(*
    MCS2 Motion Stage
    Controls a stage in CSP (NC), STEP_MODE, and Homing via DS402 interface.
    - Uses overridden Position Holding timer.
    - power enable mode must be 'DURING_MOTION' for closed-loop (CSP) control.
    - Set bServo PV to true for closed-loop, clear for open-loop (step mode).
*)
{attribute 'call_after_init'}
FUNCTION_BLOCK FB_MotionStageMCS2

VAR
    {attribute 'no_copy'}
    stMotionStage		: REFERENCE TO ST_MotionStage;
    {attribute 'no_copy'}
    stChanParams       : REFERENCE TO ST_MCS2ChanParameter;
    // Hardware I/O
    {attribute 'pytmc' := 'pv:'}
    stDS402Drive		: ST_DS402Drive;

    fbDriveManager		: FB_MCS2DriveManager;
    fbReadChanParams	: FB_ReadChanParameters;
    fbStepMode 			: FB_MCS2StepMode;
    fbhome 				: FB_MCS2Home;
    fbCalibrate			: FB_MCS2Calibrate;
    fbWriteParameters 	: FB_WriteChanParameters;
    fbReadDriveCodes 	: FB_ReadDriveCodes;

    {attribute 'hide'}
    eModule                 : E_Module;
    {attribute 'hide'}
    eDoneCause              : E_MoveDoneCause := E_MoveDoneCause.Unknown;
    {attribute 'hide'}
    fbMcPower               : MC_Power;
    {attribute 'hide'}
    fbMcMoveAbsolute        : MC_MoveAbsolute;
    {attribute 'hide'}
    fbMcHalt                : MC_Halt;
    {attribute 'hide'}
    fbMcReset               : MC_Reset;
    {attribute 'hide'}
    fbMcWriteParameter      : MC_WriteParameter;
    {attribute 'hide'}
    fbMcReadParams          : MC_ReadParameterSet;
    {attribute 'hide'}
    fParameterValue : LREAL;
    fMeasuredPos: LREAL;
    fMeasuredVelo: LREAL;
    fMeasuredAcc: LREAL;
    bLastHoltTimeOut : BOOL;
    bRestoreWaitRetry   : BOOL;
    {attribute 'hide'}
    bEnPosLag               : BOOL;
    {attribute 'hide'}
    bWrongParameter         : BOOL;
    {attribute 'hide'}
    bExecMove               : BOOL;
    {attribute 'hide'}
    bExecHome               : BOOL;
    {attribute 'hide'}
    bNewMoveReq             : BOOL;
    {attribute 'hide'}
    bPrepareDisable         : BOOL;
    {attribute 'hide'}
    bHalt                   : BOOL;
    {attribute 'hide'}
    bLimOverride            : BOOL;
    {attribute 'hide'}
    bPositionHold           : BOOL;
    {attribute 'hide'}
    bLocalExec              : BOOL;
    {attribute 'hide'}
    bSystemInit             : BOOL;
    {attribute 'hide'}
    bRestoreLoad             : BOOL;
    {attribute 'hide'}
    bExecParamRead          : BOOL;

    {attribute 'hide'}
    bRecentEnPosLagStatus    : BOOL;

    {attribute 'hide'}
    bReset                   : BOOL;
    bFault : BOOL := FALSE;
    {attribute 'hide'}
    nCmdDataLocal            : INT;
    tonHoldTime              : TON;
    {attribute 'hide'}
    NCParamsTimer            : TON;
    {attribute 'hide'}
    tonRestoreRetry          : TON;
    {attribute 'hide'}
    rtExec                   : R_TRIG;
    {attribute 'hide'}
    rtMoveCmdShortcut        : R_TRIG;
    {attribute 'hide'}
    rtHomeCmdShortcut        : R_TRIG;
    {attribute 'hide'}
    rtEnableMode             : R_TRIG;
    {attribute 'hide'}
    rtUserExec               : R_TRIG;
    {attribute 'hide'}
    rtMoveDone               : R_TRIG;
    {attribute 'hide'}
    rtNewMoveReq             : R_TRIG;
    {attribute 'hide'}
    ftExec                   : F_TRIG;
    rtHaltEdge : R_TRIG;
    {attribute 'hide'}
    rtStepCmdShortcut		 : R_TRIG;
    {attribute 'hide'}
    rtStepFwdCmdShortcut	 : R_TRIG;
    {attribute 'hide'}
    rtStepRevCmdShortcut	 : R_TRIG;
    {attribute 'hide'}
    rtCalibrateCmdShortcut	 : R_TRIG;
    {attribute 'hide'}
    tSDOOpsTimer 			 : TON;
    {attribute 'hide'}
    bParamsEnable			 : BOOL;
    {attribute 'hide'}
    bDelayReadAtInit 		 : BOOL;
    bBaseExec: BOOL;
    nCommandLocal  			 : E_MCS2OpMode := E_MCS2OpMode.CSP;
END_VAR

VAR CONSTANT
    {attribute 'hide'}
    nChanSoftLimitBase       : WORD := 16#200E;
    {attribute 'hide'}
    nChanHomeOffsetBase      : WORD := 16#607C;
    {attribute 'hide'}
    nChanHomeMethodBase      : WORD := 16#6098;
    {attribute 'hide'}
    nChanHomingSpeedBase     : WORD := 16#6099;
    {attribute 'hide'}
    nChanhomingAccBase       : WORD := 16#609A;
    {attribute 'hide'}
    nChanErrorCodeBase       : WORD := 16#603F;
    {attribute 'hide'}
    nChanFErrWinBase         : WORD := 16#6065;
    {attribute 'hide'}
    nChanOfsBase             : WORD := 16#800;      // For SmartAct MCS2 and E-727
    {attribute 'hide'}
    nChanEncErrorCode        : WORD := 16#7300;     // Motor encoder defective code (for save/restore)
    {attribute 'hide'}
    nChanSoftLimBase         : WORD := 16#200E;
    {attribute 'hide'}
    nChanOlStepBase          : WORD := 16#2022;
    {attribute 'hide'}
    nChanOlStepAmpBase       : WORD := 16#2023;
    {attribute 'hide'}
    nChanOlStepFreqBase      : WORD := 16#2024;
    {attribute 'hide'}
    nChanMaxCloseLoopFreqBase: WORD := 16#2001;
    {attribute 'hide'}
    nChanPositionerTypeBase  : WORD := 16#2000;
    {attribute 'hide'}
    nCHanCalibrationOptBase  : WORD := 16#2004;
    {attribute 'hide'}
    nChanSensorPowerModeBase : WORD := 16#2007;
    {attribute 'hide'}
    nChanReferencingOptBase  : WORD := 16#200B;
    {attribute 'hide'}
    nChanReferenceTypeBase   : WORD := 16#200A;
    {attribute 'hide'}
    nChanSafeDirBase         : WORD := 16#200C;
    {attribute 'hide'}
    nChanMotorLoadBase       : WORD := 16#200D;
    {attribute 'hide'}
    nChannelTypeBase         : WORD := 16#200F;
    {attribute 'hide'}
    nChannelStateBase        : WORD := 16#2025;
    {attribute 'hide'}
    nChanLogicalScaleOffsetBase  : WORD := 16#2008;
    {attribute 'hide'}
    nChanLogicalScaleInvBase     : WORD := 16#2009;
    {attribute 'hide'}
    nChanChannelTempBase         : WORD := 16#2026;
    {attribute 'hide'}
    nChanMovementTypeBase        : WORD := 16#2003;
    {attribute 'hide'}
    nChanBaseUnitBase            : WORD := 16#2005;
    {attribute 'hide'}
    nChanBaseResolutionBase      : WORD := 16#2006;
    {attribute 'hide'}
    nChanDistCodeInvBase         : WORD := 16#2029;
    {attribute 'hide'}
    nChanPositionerCtrlOptBase   : WORD := 16#2027;
    {attribute 'hide'}
    nChanActuatorModeBase        : WORD := 16#2028;
    {attribute 'hide'}
    nChanMotorLoadProtBase       : WORD := 16#202B;
    {attribute 'hide'}
    nChanDiagClfBase             : WORD := 16#202A;
    // Held as constants so the retract check below cannot drift from the text posted.
    {attribute 'hide'}
    sMsgPosLimit                 : STRING := 'Cannot move past positive limit.';
    {attribute 'hide'}
    sMsgNegLimit                 : STRING := 'Cannot move past Negative limit.';
END_VAR

VAR PERSISTENT
    bSaved                   : BOOL;
    fSavedPosition           : LREAL;
    bLastPositiveDirection   : BOOL;
    bLastNegativeDirection   : BOOL;
END_VAR

IF NOT __ISVALIDREF(stMotionStage)
OR NOT __ISVALIDREF(stChanParams) THEN
    RETURN;
END_IF

// When the PLC autoboots, I/O is not yet valid after 'call_after_init'
IF bSystemInit THEN
    IF stMotionStage.Axis.NcToPlc.AxisId <> 0 THEN
        bExecParamRead	:= TRUE;
        stChanParams.bStageReady  := TRUE;
        bSystemInit	:= FALSE;
        stChanParams.fPosition    := stMotionStage.Axis.NcToPlc.ActPos;
    END_IF
END_IF

(*
  Shortcut command edge detection
  Move requests can arrive via bMoveCmd (shortcut) or directly via bExecute
*)
rtMoveCmdShortcut    (CLK := stMotionStage.bMoveCmd);
rtHomeCmdShortcut    (CLK := stMotionStage.bHomeCmd);
rtStepCmdShortcut    (CLK := stChanParams.bStepMoveCmd);
rtStepFwdCmdShortcut (CLK := stChanParams.bStepForwardCmd);
rtStepRevCmdShortcut (CLK := stChanParams.bStepReverseCmd);
rtCalibrateCmdShortcut(CLK := stChanParams.bCalibrationCmd);

IF rtMoveCmdShortcut.Q AND NOT stMotionStage.bExecute THEN
    stMotionStage.bExecute := TRUE;
    stMotionStage.nCommand := E_EpicsMotorCmd.MOVE_ABSOLUTE;
    bEnPosLag              := bRecentEnPosLagStatus;
    fParameterValue        := BOOL_TO_LREAL(bRecentEnPosLagStatus);

ELSIF rtStepCmdShortcut.Q AND NOT stMotionStage.bExecute THEN
    stMotionStage.bExecute := TRUE;
    stMotionStage.nCommand := E_EpicsMotorCmd.JOG;
    bEnPosLag              := bRecentEnPosLagStatus;
    fParameterValue        := BOOL_TO_LREAL(bRecentEnPosLagStatus);

ELSIF rtStepFwdCmdShortcut.Q AND NOT stMotionStage.bExecute THEN
    // Forward jog: drive the step count positive, then step
    stChanParams.nChanStep := ABS(stChanParams.nChanStep);
    stMotionStage.bExecute := TRUE;
    stMotionStage.nCommand := E_EpicsMotorCmd.JOG;
    bEnPosLag              := bRecentEnPosLagStatus;
    fParameterValue        := BOOL_TO_LREAL(bRecentEnPosLagStatus);

ELSIF rtStepRevCmdShortcut.Q AND NOT stMotionStage.bExecute THEN
    // Reverse jog: drive the step count negative, then step
    stChanParams.nChanStep := -ABS(stChanParams.nChanStep);
    stMotionStage.bExecute := TRUE;
    stMotionStage.nCommand := E_EpicsMotorCmd.JOG;
    bEnPosLag              := bRecentEnPosLagStatus;
    fParameterValue        := BOOL_TO_LREAL(bRecentEnPosLagStatus);

ELSIF rtCalibrateCmdShortcut.Q AND NOT stMotionStage.bExecute THEN
    stMotionStage.bExecute := TRUE;
    stMotionStage.nCommand := E_EpicsMotorCmd.CALIBRATE;
    bEnPosLag              := bRecentEnPosLagStatus;
    fParameterValue        := BOOL_TO_LREAL(bRecentEnPosLagStatus);

ELSIF rtHomeCmdShortcut.Q AND NOT stMotionStage.bExecute THEN
    stMotionStage.nCommand := E_EpicsMotorCmd.HOME;
    stMotionStage.nCmdData := stChanParams.eHomeMode;
    stMotionStage.bExecute := (stChanParams.eHomeMode = E_MCS2HomeMethod.AutoMethod)
                              OR (stChanParams.eHomeMode = E_MCS2HomeMethod.CurrentPositionMethod);

    IF stMotionStage.stAxisParameters.bCtrlEnablePosDiffControl.0 THEN
        bRecentEnPosLagStatus := stMotionStage.stAxisParameters.bCtrlEnablePosDiffControl.0;
        // trigger WriteParameterNC to disable pos lag during homing
        bEnPosLag             := TRUE;
        // write 0 = disable position lag monitoring
        fParameterValue       := 0;
    END_IF
END_IF

// Main execute edge: covers both shortcut and direct bExecute paths
rtUserExec(CLK := stMotionStage.bExecute);

// Valid move request: not busy, rising execute edge, no error
bNewMoveReq S= NOT stMotionStage.bBusy AND rtUserExec.Q AND NOT stMotionStage.bError;
bNewMoveReq R= NOT stMotionStage.bExecute OR stMotionStage.bError;
bPrepareDisable R= bNewMoveReq;

IF rtUserExec.Q THEN
    //nCommandLocal := stMotionStage.nCommand;
    // Cover direct bExecute path, shortcut path already set bEnPosLag/fParameterValue
    IF NOT rtMoveCmdShortcut.Q
        AND NOT rtStepCmdShortcut.Q
        AND NOT rtCalibrateCmdShortcut.Q
    THEN
        bEnPosLag       := bRecentEnPosLagStatus;
        fParameterValue := BOOL_TO_LREAL(bRecentEnPosLagStatus);
    END_IF

    IF NOT stMotionStage.bHomeCmd
        AND NOT stChanParams.stChannelState.bIsReferenced THEN
        IF stChanParams.eHomeMode <> E_EpicsHomeCmd.NONE
            AND NOT stMotionStage.bHomed THEN
            stMotionStage.sErrorMessage := 'Axis homing mode set, but homing routine pending';
        END_IF
    END_IF
END_IF

// Drive manager
fbDriveManager(
    stMotionStage        := stMotionStage,
    stDS402Drive         := stDS402Drive,
    stMCS2ChanParameter  := stChanParams,
    bUserExec            := rtUserExec.Q,
    eRequestedManualMode => nCommandLocal
);

// Enable mode handling
rtEnableMode(CLK := (stMotionStage.nEnableMode = E_StageEnableMode.DURING_MOTION));

CASE stMotionStage.nEnableMode OF
    E_StageEnableMode.ALWAYS:
        stMotionStage.bEnable := stMotionStage.bSafetyReady;

    E_StageEnableMode.DURING_MOTION:
        IF rtEnableMode.Q THEN
            stMotionStage.bEnable := FALSE;
        END_IF
        IF bNewMoveReq THEN
            bPositionHold        := FALSE;
            tonHoldTime.IN       := FALSE;
            stMotionStage.bEnable:= stMotionStage.bSafetyReady;
            bLastHoltTimeOut     := FALSE;
            bHalt                := FALSE;
        END_IF
END_CASE

// Interlock: Reacts on internal limit conditions
Interlock();

bBaseExec := NOT stMotionStage.bError
             AND stMotionStage.bExecute
             AND stMotionStage.bAllEnable
             AND stMotionStage.bSafetyReady;

IF fbDriveManager.bCSPModeEnabled THEN
    // Close loop: gate on NC standstill state (bEnableDone)
    bLocalExec := bBaseExec
                  AND stMotionStage.bEnableDone
                  AND stMotionStage.nCommand = E_EpicsMotorCmd.MOVE_ABSOLUTE;

ELSIF fbDriveManager.bHomeModeEnabled THEN
    // Open loop homing: gate on DS402 operational state
    bLocalExec := bBaseExec
                  AND fbDriveManager.bOperational
                  AND stMotionStage.nCommand = E_EpicsMotorCmd.HOME;

ELSIF fbDriveManager.bStepModeEnabled THEN
    // Open loop step: gate on DS402 operational state
    bLocalExec := bBaseExec
                  AND fbDriveManager.bOperational
                  AND stMotionStage.nCommand = E_EpicsMotorCmd.JOG;

ELSIF fbDriveManager.bCalibrationModeEnabled THEN
    // Open loop calibration: gate on DS402 operational state
    bLocalExec := bBaseExec
                  AND fbDriveManager.bOperational
                  AND stMotionStage.nCommand = E_EpicsMotorCmd.CALIBRATE;
ELSE
    bLocalExec := FALSE;
END_IF

bExecMove := bLocalExec AND ((stMotionStage.nCommand = E_EpicsMotorCmd.MOVE_ABSOLUTE)
                          OR  (stMotionStage.nCommand = E_EpicsMotorCmd.JOG)
                          OR  (stMotionStage.nCommand = E_EpicsMotorCmd.CALIBRATE));
bExecHome := bLocalExec AND NOT bExecMove;

rtExec(CLK := bLocalExec);
IF rtExec.Q THEN
    stDS402Drive.nDriveControl.8 := FALSE;
    stMotionStage.bDone          := FALSE;
END_IF


IF NOT fbDriveManager.bDS402Manual THEN
    stMotionStage.Axis.ReadStatus();
END_IF

// Get definitive bEnableDone from NC axis state
CASE stMotionStage.Axis.Status.MotionState OF
    MC_AXISSTATE_UNDEFINED, MC_AXISSTATE_DISABLED, MC_AXISSTATE_ERRORSTOP:
        stMotionStage.bEnableDone := FALSE;
    ELSE
        stMotionStage.bEnableDone := TRUE;
END_CASE

// Reset handling
IF stMotionStage.bReset THEN
    stMotionStage.bExecute          := FALSE;
    stMotionStage.bError            := FALSE;
    stMotionStage.nErrorId          := 0;
    stMotionStage.sErrorMessage     := '';
    stMotionStage.sCustomErrorMessage := '';
    fbStepMode.Reset();
    fbhome.Reset();
    bReset := TRUE;
    IF fbDriveManager.bDS402Manual THEN
        stDS402Drive.nDriveControl.7 := TRUE;
    END_IF
    stMotionStage.bReset := FALSE;
END_IF

// Stop/halt detection. bHalt is the user-stop channel only: execute dropped
// mid-move. Limit reaction is handled by the direction enables, not from here.
ftExec(CLK := stMotionStage.bExecute);
bHalt := ftExec.Q AND stMotionStage.bBusy;
rtHaltEdge(CLK := bHalt);
IF rtHaltEdge.Q AND fbDriveManager.bDS402Manual THEN
    fbStepMode.Halt();
    fbhome.Halt();
    stDS402Drive.nDriveControl.8 := TRUE;
END_IF

WriteParameterNC(
    Execute         := bEnPosLag,
    ParameterNumber := MC_AxisParameter.AxisEnPositionLagMonitoring,
    ParameterValue  := fParameterValue
);

bParamsEnable := stMotionStage.bAxisParamsInit AND stChanParams.bEnableHardwareOps;

fbWriteParameters(
    bEnable             := bParamsEnable,
    bErrorAcknowledge   := stMotionStage.bReset,
    stDS402Drive        := stDS402Drive,
    stMotionStage       := stMotionStage,
    stChanParams := stChanParams
);

CASE nCommandLocal OF
    E_MCS2OpMode.CSP:
        Reset();
        Power();
        Halt();
        (*Wait for drive to be in the correct mode after a request was validated *)
        MoveAbsolute();
        (*
          IN CSP mode the drive control word is update via the NC
          Manual step mode and Homing will override this
        *)

        stDS402Drive.nModeOfOperation := stDS402Drive.nModeOfOperationNC;
        stDS402Drive.nDriveControl    := stDS402Drive.nDriveControlNC;

    E_MCS2OpMode.HOME:
        (*DS402 Manual Homing*)
        fbhome(
            bExecute := bExecHome AND fbWriteParameters.bParamsSet,
            stDS402Drive  := stDS402Drive,
            stMotionStage := stMotionStage
        );

    E_MCS2OpMode.STEP:
        fbStepMode(
            bExecute       := bExecMove AND fbWriteParameters.bParamsSet,
            stDS402Drive  := stDS402Drive,
            stMotionStage := stMotionStage
        );

    E_MCS2OpMode.CALIBRATE:
        fbCalibrate(
            bExecute	 := bExecMove AND fbWriteParameters.bParamsSet,
            stDS402Drive  := stDS402Drive,
            stMotionStage := stMotionStage
        );
END_CASE

stMotionStage.bBusy := fbMcMoveAbsolute.Busy
                       OR stChanParams.stChannelState.bReferencing
                       OR fbStepMode.bStepMoveBusy
                       OR stChanParams.stChannelState.bCalibrating;
// Check done moving via user stop, limit hit, Target Position reached, or from homing.
PostMoveChecks();
// update encoder value and calibrated position
ScaleEncRawValue();
// Drive parameters
ExposedParameters(Enable := stChanParams.bStageReady, tRefreshDelay := T#2S);
// Read MCS2 Channel Parameters
fbReadChanParams(
    bEnable             := bParamsEnable,
    stMotionStage       := stMotionStage,
    stMCS2ChanParameter := stChanParams,
    stDS402Drive        := stDS402Drive,
);
(* Save and restore as long as not an absolute encoder*)
PersistParameters(Enable := stChanParams.bStageReady);
(*Restore encoder value at initialization*)
RestoreMotionParams(Enable := stChanParams.bStageReady);
(*EPICS Motor record Update*)
UpdateEpicsStatus();

(*
    Error from functions and Nc. The error will send to EPICS interface based on predifined
    priority: axis, power, backlash, absoluteMove, etc...
*)
IF fbMcPower.Error AND fbMcPower.Active THEN
    stMotionStage.bError   := fbMcPower.Error;
    stMotionStage.nErrorId := fbMcPower.ErrorID;
ELSIF fbMcMoveAbsolute.Error THEN
    stMotionStage.bError   := fbMcMoveAbsolute.Error;
    stMotionStage.nErrorId := fbMcMoveAbsolute.ErrorID;
ELSIF fbMcHalt.Error AND fbMcHalt.Active THEN
    stMotionStage.bError   := fbMcHalt.Error;
    stMotionStage.nErrorId := fbMcHalt.ErrorID;
ELSIF fbMcReset.Error THEN
    stMotionStage.bError   := fbMcReset.Error;
    stMotionStage.nErrorId := fbMcReset.ErrorID;
ELSIF fbMcWriteParameter.Error THEN
    stMotionStage.bError   := fbMcWriteParameter.Error;
    stMotionStage.nErrorId := fbMcWriteParameter.ErrorID;
ELSIF fbMcReadParams.Error AND NOT stMotionStage.bBusy THEN
    stMotionStage.bError   := fbMcReadParams.Error;
    stMotionStage.nErrorId := fbMcReadParams.ErrorID;
ELSE
    IF stMotionStage.bBusy THEN
        // Clear the display message during normal motion, but leave sCustomErrorMessage
        // intact: Interlock may have just set it on this same cycle, and the NC error
        // that latches bError will not be visible until the next cycle.
        stMotionStage.sErrorMessage := '';
    END_IF
END_IF

(*Double function, prioritize NC error otherwise read drive channel error code*)
fbReadDriveCodes(
    bEnable             := bParamsEnable,
    stMotionStage       := stMotionStage,
    stMCS2ChanParameter := stChanParams,
    stDS402Drive        := stDS402Drive,
);

IF stMotionStage.sCustomErrorMessage <> ''
    AND stMotionStage.sErrorMessage = '' THEN
    stMotionStage.sErrorMessage := stMotionStage.sCustomErrorMessage;
END_IF

(*Clear motion flag when error occurs*)
IF stMotionStage.bError THEN
    stMotionStage.bExecute := FALSE;
    stMotionStage.bBusy    := FALSE;
    stMotionStage.bDone    := FALSE;
    stMotionStage.bEnable  := FALSE;
END_IF

(* We've got the rising edge clear these flags.*)
stMotionStage.bMoveCmd             := FALSE;
stMotionStage.bHomeCmd             := FALSE;
stChanParams.bStepMoveCmd   := FALSE;
stChanParams.bStepForwardCmd := FALSE;
stChanParams.bStepReverseCmd := FALSE;
stChanParams.bCalibrationCmd := FALSE;

METHOD PUBLIC  ExposedParameters
VAR_INPUT
    Enable : BOOL;
    tRefreshDelay: TIME;
END_VAR

VAR_INST
    {attribute 'hide'}
    bParamReadTimer     : BOOL := TRUE;
END_VAR
// Periodic update of NC parameters
NCParamsTimer( IN:=Enable AND NOT bExecParamRead, PT:=tRefreshDelay);
bExecParamRead S= NCParamsTimer.Q;
fbMcReadParams(
    Parameter:= stMotionStage.stAxisParameters,
    Axis:= stMotionStage.Axis,
    Execute:= bExecParamRead );

// Copy axis parameters that we want to expose to the EPICS layer.
 stMotionStage.stAxisParametersExposed.bCtrlEnablePosDiffControl     :=  stMotionStage.stAxisParameters.bCtrlEnablePosDiffControl;
 stMotionStage.stAxisParametersExposed.bEncEnableSoftEndMaxControl   :=  stMotionStage.stAxisParameters.bEncEnableSoftEndMaxControl;
 stMotionStage.stAxisParametersExposed.bEncEnableSoftEndMinControl   :=  stMotionStage.stAxisParameters.bEncEnableSoftEndMinControl;
 stMotionStage.stAxisParametersExposed.fAccelerationMax              :=  stMotionStage.stAxisParameters.fAccelerationMax;
 stMotionStage.stAxisParametersExposed.fCtrlPosDiffMax               :=  stMotionStage.stAxisParameters.fCtrlPosDiffMax;
 stMotionStage.stAxisParametersExposed.fCtrlPosDiffMaxTime           :=  stMotionStage.stAxisParameters.fCtrlPosDiffMaxTime;
 stMotionStage.stAxisParametersExposed.fDecelerationMax              :=  stMotionStage.stAxisParameters.fDecelerationMax;
 stMotionStage.stAxisParametersExposed.fEncSoftEndMax                :=  stMotionStage.stAxisParameters.fEncSoftEndMax;
 stMotionStage.stAxisParametersExposed.fEncSoftEndMin                :=  stMotionStage.stAxisParameters.fEncSoftEndMin;
 stMotionStage.stAxisParametersExposed.fVeloMaximum                  :=  stMotionStage.stAxisParameters.fVeloMaximum;
 stMotionStage.stAxisParametersExposed.fEncOffset                       :=  stMotionStage.stAxisParameters.fEncOffset;
 stMotionStage.stAxisParametersExposed.fEncScaleFactorInternal       :=  stMotionStage.stAxisParameters.fEncScaleFactorInternal;

bExecParamRead R= fbMcReadParams.Done OR fbMcReadParams.Error;
 stMotionStage.bAxisParamsInit S= fbMcReadParams.Done;
END_METHOD

//FB_Init is always available implicitly and it is used primarily for initialization.
//The return value is not evaluated. For a specific influence, you can also declare the
//methods explicitly and provide additional code there with the standard initialization
//code. You can evaluate the return value.
METHOD FB_Init: BOOL
VAR_INPUT
    bInitRetains: BOOL; // TRUE: the retain variables are initialized (reset warm / reset cold)
    bInCopyCode: BOOL;  // TRUE: the instance will be copied to the copy code afterward (online change)
    stMotionStage	: REFERENCE TO ST_MotionStage;
    stMCS2ChanParameter : REFERENCE TO ST_MCS2ChanParameter;
    (*Mandatory must be unique for each MCS2 axis *)
    eModule : E_Module;
END_VAR
THIS^.stMotionStage REF= stMotionStage;
THIS^.stChanParams REF= stMCS2ChanParameter;
THIS^.eModule := eModule;
END_METHOD

METHOD Halt
fbMcHalt(
    Axis :=  stMotionStage.Axis,
    Execute := bHalt,
    Deceleration :=  stMotionStage.fDeceleration,
    BufferMode := MC_BufferMode.MC_Aborting,
);
IF fbMcHalt.Done THEN
    bHalt := FALSE;
END_IF
END_METHOD

METHOD PUBLIC Interlock

VAR_INST
    {attribute 'hide'}
    bPositiveDirection  : BOOL;
    {attribute 'hide'}
    bNegativeDirection  : BOOL;
    {attribute 'hide'}
    ftForwardEnabled    : F_TRIG;
    {attribute 'hide'}
    ftBackwardEnabled   : F_TRIG;
    {attribute 'hide'}
    bHitForwardLimit    : BOOL;
    {attribute 'hide'}
    bHitBackwardLimit   : BOOL;
    {attribute 'hide'}
    fCurrentPosition    : LREAL;
END_VAR
// Positive or Negative direction.
// In step mode fPosDiff is unreliable for direction: fPosition is the stale NC setpoint
// and fMeasuredPos is the live encoder, so their difference inverts as the motor moves.
// Use the step count sign instead, which is set explicitly at command issue time.
IF fbDriveManager.bStepModeEnabled THEN
    bPositiveDirection := stMotionStage.bBusy AND stChanParams.nChanStep > 0;
    bNegativeDirection := stMotionStage.bBusy AND stChanParams.nChanStep < 0;
ELSE
    bPositiveDirection := stMotionStage.bBusy AND stMotionStage.fPosDiff > 0;
    bNegativeDirection := stMotionStage.bBusy AND stMotionStage.fPosDiff < 0;
END_IF

// If the drive starts limited and no direction history is available, infer the
// blocked side from the nearest configured software range limit. The aggregate
// InternalLimitActive bit does not identify the side by itself.
fCurrentPosition := DINT_TO_LREAL(stMotionStage.nRawEncoderDINT)
                    * MAX(stMotionStage.stAxisParameters.fEncScaleFactorInternal,
                          stChanParams.fScalingFactor);
IF stDS402Drive.stDriveStatus.InternalLimitActive THEN
    IF NOT bLastPositiveDirection AND NOT bLastNegativeDirection THEN
        IF fbReadChanParams.bAllReadsComplete THEN
            IF stChanParams.nSoftLimMax > stChanParams.nSoftLimMin THEN
                IF ABS(fCurrentPosition - stChanParams.nSoftLimMin)
                   < ABS(stChanParams.nSoftLimMax - fCurrentPosition) THEN
                    bLastNegativeDirection := TRUE;
                ELSE
                    bLastPositiveDirection := TRUE;
                END_IF
            END_IF
        END_IF
    END_IF
END_IF

// Preserve the last commanded direction across the stop and PLC restart. The
// drive exposes one aggregate limit bit, so this retained context identifies
// which direction should remain blocked during recovery.
IF NOT stDS402Drive.stDriveStatus.InternalLimitActive
    OR (NOT bHitForwardLimit AND NOT bHitBackwardLimit) THEN
    IF bPositiveDirection THEN
        bLastPositiveDirection := TRUE;
        bLastNegativeDirection := FALSE;
    ELSIF bNegativeDirection THEN
        bLastPositiveDirection := FALSE;
        bLastNegativeDirection := TRUE;
    END_IF
END_IF

// Latch which physical limit was hit; clear once the drive is no longer reporting a limit.
// A single InternalLimitActive bit covers both directions, so direction at the time of
// the hit is used to determine which enable to hold off.
bHitForwardLimit  S= stDS402Drive.stDriveStatus.InternalLimitActive
                   AND (bPositiveDirection OR bLastPositiveDirection);
bHitBackwardLimit S= stDS402Drive.stDriveStatus.InternalLimitActive
                    AND (bNegativeDirection OR bLastNegativeDirection);
bHitForwardLimit  R= NOT stDS402Drive.stDriveStatus.InternalLimitActive;
bHitBackwardLimit R= NOT stDS402Drive.stDriveStatus.InternalLimitActive;

// An active limit with no known direction disables both directions. Once the
// hit direction is known, only that direction is disabled for reverse recovery.
stMotionStage.bLimitForwardEnable := NOT stDS402Drive.stDriveStatus.InternalLimitActive
                                     OR (bHitBackwardLimit AND NOT bHitForwardLimit);
stMotionStage.bLimitBackwardEnable := NOT stDS402Drive.stDriveStatus.InternalLimitActive
                                      OR (bHitForwardLimit AND NOT bHitBackwardLimit);

// use falling trigger to avoid spamming sErrorMessage
ftForwardEnabled(CLK := stMotionStage.bLimitForwardEnable);
ftBackwardEnabled(CLK := stMotionStage.bLimitBackwardEnable);

// A limit hit is the lowest priority message. Never post one over a latched fault,
// and retract our own once the drive releases the limit so a stale warning cannot
// later be promoted into sErrorMessage. The drive stops the positioner itself and
// SetEnables drops the offending direction, so no halt is requested here.
IF NOT stMotionStage.bError AND NOT fbhome.bHomeMoveBusy THEN
    IF bHitForwardLimit AND ftForwardEnabled.Q THEN
        stMotionStage.sCustomErrorMessage := sMsgPosLimit;
    ELSIF bHitBackwardLimit AND ftBackwardEnabled.Q THEN
        stMotionStage.sCustomErrorMessage := sMsgNegLimit;
    END_IF
END_IF

IF NOT bHitForwardLimit AND NOT bHitBackwardLimit
   AND (stMotionStage.sCustomErrorMessage = sMsgPosLimit
        OR stMotionStage.sCustomErrorMessage = sMsgNegLimit) THEN
    stMotionStage.sCustomErrorMessage := '';
END_IF

IF NOT  stMotionStage.bError AND  stMotionStage.bExecute AND NOT  stMotionStage.bUserEnable THEN
     stMotionStage.bError := TRUE;
     stMotionStage.nErrorId := 1;
     stMotionStage.sCustomErrorMessage := 'Move requested, but user enable is disabled!';
END_IF

// Update all enable booleans
SetEnables();
END_METHOD

METHOD PUBLIC  MoveAbsolute
fbMcMoveAbsolute(
    Axis :=  stMotionStage.Axis,
    Execute := bExecMove AND fbMcPower.Status AND fbDriveManager.bCSPModeEnabled,
    Position :=  stMotionStage.fPosition,
    Velocity :=  stMotionStage.fVelocity,
    Acceleration :=  stMotionStage.fAcceleration,
    Deceleration :=  stMotionStage.fDeceleration,
    BufferMode := MC_BufferMode.MC_Aborting,
);

IF fbMcMoveAbsolute.Done (*OR fbMcReset.Done*) THEN
    (*Hold the position in close loop before dropping power, a positional drift will occur then*)
    IF ( stMotionStage.nEnableMode = E_StageEnableMode.DURING_MOTION ) THEN
        bPositionHold := TRUE;
        tonHoldTime.IN:=TRUE;
    END_IF
END_IF
END_METHOD

METHOD PersistParameters
VAR_INPUT
    Enable  : BOOL;
END_VAR

VAR_INST
    {attribute 'hide'}
    bEncError           : BOOL;
END_VAR
// Save Encoder position
// needs some pre-conditions to use persistent storage
IF Enable THEN
    // Check ST_MotionStage for an encoder error (range 0x44nn)
    bEncError:=  stMotionStage.Axis.Status.Error AND  (  stMotionStage.Axis.Status.ErrorID  >= 16#4400  AND  stMotionStage.Axis.Status.ErrorID <= 16#44FF );
    // Do not save if we're currently loading or if there is an encoder error
    IF NOT bRestoreLoad AND NOT bEncError AND NOT bRestoreWaitRetry THEN
        fSavedPosition :=  stMotionStage.Axis.NcToPlc.ActPos;
        // This persistent variable lets us check if anything was saved
        // It will be TRUE at startup if we have saved values
        bSaved := TRUE;
    END_IF
END_IF
END_METHOD

{attribute 'call_after_init'}
(*  eModule: Mandatory must be unique for each MCS2 axis
    clears startup errors or warnings. the process is completed at run time
    SDO update of Drive and open Loop parameter Indexes based on module number
*)
METHOD PostInit
(* SDO update of Drive and open Loop parameter Indexes based on module number *)
stChanParams.nChanErrorCodeIdx        	:= nChanErrorCodeBase         	+ ((eModule-1) * nChanOfsBase);
stChanParams.nChanFErrWinIdx          	:= nChanFErrWinBase           	+ ((eModule-1) * nChanOfsBase);
stChanParams.nChanSoftLimitIdx        	:= nChanSoftLimitBase     		+ ((eModule-1) * nChanOfsBase);
stChanParams.nChanHomeOffsIdx         	:= nChanHomeOffsetBase        	+ ((eModule-1) * nChanOfsBase);
stChanParams.nChanHomeMethodIdx         := nChanHomeMethodBase       	+ ((eModule-1) * nChanOfsBase);
stChanParams.nChanHomeVeloIdx         	:= nChanHomingSpeedBase       	+ ((eModule-1) * nChanOfsBase);
stChanParams.nChanhomeAccIdx          	:= nChanhomingAccBase         	+ ((eModule-1) * nChanOfsBase);
stChanParams.nChanStepIdx             	:= nChanOlStepBase            	+ ((eModule-1) * nChanOfsBase);
stChanParams.nChanStepFreqIdx         	:= nChanOlStepFreqBase        	+ ((eModule-1) * nChanOfsBase);
stChanParams.nChanStepAmpIdx          	:= nChanOlStepAmpBase         	+ ((eModule-1) * nChanOfsBase);
stChanParams.nChanMaxCloseLoopFreqIdx   := nChanMaxCloseLoopFreqBase  	+ ((eModule-1) * nChanOfsBase);
stChanParams.nChanPositionerTypeIdx     := nChanPositionerTypeBase    	+ ((eModule-1) * nChanOfsBase);
stChanParams.nChanCalibrationOptIdx     := nCHanCalibrationOptBase    	+ ((eModule-1) * nChanOfsBase);
stChanParams.nChanSensorPowerModeIdx    := nChanSensorPowerModeBase   	+ ((eModule-1) * nChanOfsBase);
stChanParams.nChanReferencingOptIdx     := nChanReferencingOptBase    	+ ((eModule-1) * nChanOfsBase);
stChanParams.nChanReferenceTypeIdx      := nChanReferenceTypeBase     	+ ((eModule-1) * nChanOfsBase);
stChanParams.nChanSafeDirIdx            := nChanSafeDirBase           	+ ((eModule-1) * nChanOfsBase);
stChanParams.nChanMotorLoadIdx          := nChanMotorLoadBase         	+ ((eModule-1) * nChanOfsBase);
stChanParams.nChannelTypeIdx          	:= nChannelTypeBase       		+ ((eModule-1) * nChanOfsBase);
stChanParams.nChanStateIdx         		:= nChannelStateBase      		+ ((eModule-1) * nChanOfsBase);
stChanParams.nChanLogicalScaleOfsIdx   	:= nChanLogicalScaleOffsetBase	+ ((eModule-1) * nChanOfsBase);
stChanParams.nChanLogicalScaleInvIdx    := nChanLogicalScaleInvBase   	+ ((eModule-1) * nChanOfsBase);
stChanParams.nChanChannelTempIdx        := nChanChannelTempBase       	+ ((eModule-1) * nChanOfsBase);
stChanParams.nChanMovementTypeIdx       := nChanMovementTypeBase      	+ ((eModule-1) * nChanOfsBase);
stChanParams.nChanBaseUnitIdx           := nChanBaseUnitBase          	+ ((eModule-1) * nChanOfsBase);
stChanParams.nChanBaseResolutionIdx     := nChanBaseResolutionBase    	+ ((eModule-1) * nChanOfsBase);
stChanParams.nChanDistCodeInvIdx        := nChanDistCodeInvBase       	+ ((eModule-1) * nChanOfsBase);
stChanParams.nChanPositionerCtrlOptIdx  := nChanPositionerCtrlOptBase 	+ ((eModule-1) * nChanOfsBase);
stChanParams.nChanActuatorModeIdx       := nChanActuatorModeBase      	+ ((eModule-1) * nChanOfsBase);
stChanParams.nChanMotorLoadProtIdx      := nChanMotorLoadProtBase     	+ ((eModule-1) * nChanOfsBase);
stChanParams.nChanDiagClfIdx            := nChanDiagClfBase           	+ ((eModule-1) * nChanOfsBase);
bSystemInit := TRUE;
END_METHOD

METHOD PRIVATE PostMoveChecks : BOOL
VAR_INST
    rtAbortedHome        : R_TRIG;
    rtAbortedStepMove    : R_TRIG;
    rtAbortedCalibration : R_TRIG;
    rtResetDone          : R_TRIG;
    rtHaltDone           : R_TRIG;
    rtMoveDone           : R_TRIG;
    rtHomeDone           : R_TRIG;
    rtStepMoveDone       : R_TRIG;
    rtCalibrationDone    : R_TRIG;
    ftEnableFallEdge     : F_TRIG;
END_VAR
rtAbortedHome(CLK := fbhome.bHomeMoveAborted);
rtAbortedStepMove(CLK := fbStepMode.bStepMoveAborted);
rtAbortedCalibration(CLK := fbCalibrate.bCalibrateMoveAborted);

rtResetDone(CLK := fbMcReset.Done);
rtHaltDone(CLK := fbMcHalt.Done);

rtMoveDone(CLK := fbMcMoveAbsolute.Done);
rtHomeDone(CLK := fbhome.bHomeMoveDone);
rtStepMoveDone(CLK := fbStepMode.bStepMoveDone);
rtCalibrationDone(CLK := fbCalibrate.bCalibrateMoveDone);

IF rtAbortedHome.Q OR rtAbortedStepMove.Q OR rtAbortedCalibration.Q
   OR rtResetDone.Q OR rtHaltDone.Q
   OR rtMoveDone.Q OR rtHomeDone.Q OR rtStepMoveDone.Q OR rtCalibrationDone.Q THEN

    IF NOT stMotionStage.bDone THEN
        stMotionStage.bExecute := FALSE;;
        stMotionStage.bHomed := fbhome.bHomeMoveDone;
        IF rtMoveDone.Q THEN
            stMotionStage.bDone := TRUE;
            eDoneCause := E_MoveDoneCause.MoveDone;
        ELSIF rtStepMoveDone.Q THEN
            stMotionStage.bDone := TRUE;
            eDoneCause := E_MoveDoneCause.StepMoveDone;
        ELSIF rtHomeDone.Q THEN
            stMotionStage.bDone := TRUE;
            eDoneCause := E_MoveDoneCause.HomeDone;
            // Homing runs in DS402 manual HOME mode. Request closed-loop so the
            // drive manager switches the drive back to CSP now that homing is done.
            stChanParams.eOpModeReq := E_MCS2OpModeReq.CLOSED_LOOP;
        ELSIF rtCalibrationDone.Q THEN
            stMotionStage.bDone := TRUE;
            eDoneCause := E_MoveDoneCause.CalibrationDone;
            // Calibration runs in DS402 manual CALIBRATE mode. Request closed-loop so
            // the drive manager switches the drive back to CSP now that calibration is done.
            stChanParams.eOpModeReq := E_MCS2OpModeReq.CLOSED_LOOP;
        ELSIF rtResetDone.Q THEN
            stMotionStage.bDone := TRUE;
            eDoneCause := E_MoveDoneCause.ResetDone;
        ELSIF rtHaltDone.Q THEN
            stMotionStage.bDone := TRUE;
            eDoneCause := E_MoveDoneCause.HaltDone;
        ELSIF rtAbortedHome.Q THEN
            stMotionStage.bDone := TRUE;
            eDoneCause := E_MoveDoneCause.AbortedHome;
        ELSIF rtAbortedStepMove.Q THEN
            stMotionStage.bDone := TRUE;
            eDoneCause := E_MoveDoneCause.AbortedStepMove;
        ELSIF rtAbortedCalibration.Q THEN
            stMotionStage.bDone := TRUE;
            eDoneCause := E_MoveDoneCause.AbortedCalibration;
        END_IF
        IF fbDriveManager.bDS402Manual THEN
            bEnPosLag := FALSE;
        END_IF
        IF (stMotionStage.nEnableMode = E_StageEnableMode.DURING_MOTION) THEN
            bPositionHold := TRUE;
            tonHoldTime.IN := TRUE;
        END_IF
        // get stable current position storage
        stChanParams.fPosition := stMotionStage.fPosition;
    END_IF
END_IF

tonHoldTime(PT := UDINT_TO_TIME(stChanParams.nHoldTime));
IF tonHoldTime.Q THEN
    bPositionHold := FALSE;
    tonHoldTime.IN := FALSE;
    bLastHoltTimeOut := TRUE;
END_IF

(* updated axis status
   Not needed in manual mode *)
IF NOT fbDriveManager.bDS402Manual THEN
     stMotionStage.Axis.ReadStatus();
END_IF

bPrepareDisable S= (stMotionStage.nEnableMode = E_StageEnableMode.DURING_MOTION) AND ftExec.Q;

IF bPrepareDisable AND fbDriveManager.bCSPModeEnabled THEN
    IF stMotionStage.Axis.Status.StandStill THEN
        IF NOT bPositionHold THEN
            bPrepareDisable := FALSE;
            stMotionStage.bEnable := FALSE; // TwinCAT NC disables MC_Power (CSP)
        END_IF
    END_IF
ELSIF bPrepareDisable AND fbDriveManager.bDS402Manual THEN
    IF fbDriveManager.bOperational THEN
        IF NOT bPositionHold THEN
            bPrepareDisable := FALSE;
            stMotionStage.bEnable := FALSE; // Manual disables via drive control word
        END_IF
    END_IF
END_IF

ftEnableFallEdge(CLK := stMotionStage.bEnable);
IF ftEnableFallEdge.Q THEN
    IF fbDriveManager.bDS402Manual THEN
        stDS402Drive.nDriveControl := 6; // Manual mode power off
    END_IF
END_IF
END_METHOD

METHOD Power
fbMcPower(
    Axis :=  stMotionStage.Axis,
    Enable :=  stMotionStage.bAllEnable,
    Enable_Positive :=  stMotionStage.bAllForwardEnable AND stChanParams.bOverrideDirEnable,
    Enable_Negative :=  stMotionStage.bAllBackwardEnable AND stChanParams.bOverrideDirEnable,
    Override := 100.0,
    BufferMode := MC_BufferMode.MC_Aborting
);
END_METHOD

METHOD Reset
fbMcReset(
    Axis :=  stMotionStage.Axis,
    Execute := bReset
);
IF fbMcReset.Done THEN
    bReset := FALSE;
END_IF
END_METHOD

METHOD RestoreMotionParams
VAR_INPUT
    Enable  : BOOL;
END_VAR

VAR_INST
    fbSetPos            : MC_SetPosition;
    {attribute 'hide'}
    bLoad               : BOOL;
    {attribute 'hide'}
    bRestoreInit        : BOOL;
    {attribute 'hide'}
    nMaxRetries         : UINT := 10;
    {attribute 'hide'}
    nCurrTries          : UINT := 0;
    {attribute 'hide'}
    nLatchError         : UDINT;
END_VAR
IF Enable THEN
    // Trigger a load if anything was saved at all
    IF NOT bRestoreInit THEN
        bRestoreInit := TRUE;
        bRestoreLoad S= bSaved;
        fbSetPos.Options.ClearPositionLag := TRUE;
    END_IF

    // Set our position if bRestoreLoad is true
    fbSetPos( Axis:= stMotionStage.Axis, Execute:=bRestoreLoad, Position:=fSavedPosition);

    IF fbSetPos.Error THEN
        // Keep the error latched, it can disappear if Execute is set to FALSE
        nLatchError := fbSetPos.ErrorID;
        nCurrTries := nCurrTries + 1;
        IF nCurrTries >= nMaxRetries THEN
        // Alert the user that something has gone wrong
         stMotionStage.bError := TRUE;
         stMotionStage.nErrorId := nLatchError;
         stMotionStage.sCustomErrorMessage := 'Error loading previously saved position.';
        ELSE
            // Reset the FB for the next retry
            fbSetPos( Axis:= stMotionStage.Axis, Execute:=bRestoreLoad, Position:=fSavedPosition);
            // Try again
            bRestoreWaitRetry := TRUE;
        END_IF
    ELSIF fbSetPos.Done THEN
         stMotionStage.fPosition := fSavedPosition;
         stMotionStage.bRestoreDone := TRUE;
    END_IF

    // Only load once, at startup
    bRestoreLoad R= fbSetPos.Done OR fbSetPos.Error;

    tonRestoreRetry( IN := bRestoreWaitRetry, PT := T#100MS);
    bRestoreLoad S= tonRestoreRetry.Q;
    bRestoreWaitRetry R= tonRestoreRetry.Q;
END_IF
END_METHOD

METHOD ScaleEncRawValue
VAR_INPUT
  //  bEnable: BOOL;
END_VAR
(* SmartACT: The encoder count from the Piezo drive is not a raw count from the embeded actuator device
   we get a calibrated nm value. thus the use of abs() since this value is signed.*)

stMotionStage.nEncoderCount:=DINT_TO_UDINT(ABS( stMotionStage.nRawEncoderDINT));

// calibrated encoder readback
IF NOT fbDriveManager.bStepModeEnabled THEN
    // Close loop NC
    fMeasuredPos:= stMotionStage.Axis.NcToPlc.ActPos;
    fMeasuredVelo := stMotionStage.Axis.NcToPlc.ActVelo;
    fMeasuredAcc :=  stMotionStage.Axis.NcToPlc.ActAcc;
    stMotionStage.fPosDiff:= stMotionStage.Axis.NcToPlc.PosDiff;
ELSE
    fMeasuredPos:=DINT_TO_REAL( stMotionStage.nRawEncoderDINT) * MAX( stMotionStage.stAxisParameters.fEncScaleFactorInternal, stChanParams.fScalingFactor);
    stMotionStage.fPosDiff:= stMotionStage.fPosition - fMeasuredPos;
    // NB: Not actual in open loop
    fMeasuredVelo := stMotionStage.fVelocity;
    fMeasuredAcc :=  stMotionStage.fAcceleration;
END_IF
END_METHOD

METHOD SetEnables
VAR_INPUT
END_VAR
 stMotionStage.bAllForwardEnable:= stMotionStage.bLimitForwardEnable
                                    AND ( stMotionStage.bGantryForwardEnable OR NOT  stMotionStage.bGantryAxis)
                                    AND  stMotionStage.stEPSForwardEnable.bEPS_OK
                                    AND  stChanParams.bOverrideDirEnable;
 stMotionStage.bAllBackwardEnable:= stMotionStage.bLimitBackwardEnable
                                    AND ( stMotionStage.bGantryBackwardEnable OR NOT  stMotionStage.bGantryAxis)
                                    AND  stMotionStage.stEPSBackwardEnable.bEPS_OK
                                    AND  stChanParams.bOverrideDirEnable;

 stMotionStage.bAllEnable:= stMotionStage.bEnable
                            AND  stMotionStage.bHardwareEnable
                            AND  stMotionStage.stEPSPowerEnable.bEPS_OK;
 stMotionStage.bAllEnable R= NOT  stMotionStage.bUserEnable;
END_METHOD

METHOD UpdateEpicsStatus
VAR_INPUT
END_VAR
//////////////////////////////////////////////////////////////////
// Transfer NC parameter status to EPICS
//////////////////////////////////////////////////////////////////
 stMotionStage.nMotionAxisID :=  stMotionStage.Axis.NcToPlc.AxisId;
 stMotionStage.stAxisStatus.bEnable:= stMotionStage.bAllEnable;
 stMotionStage.stAxisStatus.bEnabled:= stMotionStage.bEnableDone; // account for PowerEnable from power block
 stMotionStage.stAxisStatus.bError:= stMotionStage.bError;
 stMotionStage.stAxisStatus.bHomeSensor:= stMotionStage.bHome;
 stMotionStage.stAxisStatus.bLimitBwd:= stMotionStage.bAllBackwardEnable;
 stMotionStage.stAxisStatus.bLimitFwd:= stMotionStage.bAllForwardEnable;
 stMotionStage.stAxisStatus.bReset:= stMotionStage.bReset;
 stMotionStage.stAxisStatus.fAcceleration:=fMeasuredAcc;
 stMotionStage.stAxisStatus.fActDiff:= stMotionStage.fPosDiff;
 stMotionStage.stAxisStatus.fActPosition:=fMeasuredPos;
 stMotionStage.stAxisStatus.fActVelocity:=fMeasuredVelo;
 stMotionStage.stAxisStatus.fDeceleration:=fMeasuredAcc;
 stMotionStage.stAxisStatus.fOverride:=fbMcPower.Override;
 stMotionStage.stAxisStatus.fPosition:= stMotionStage.fPosition;
 stMotionStage.stAxisStatus.fVelocity:= stMotionStage.fVelocity;
 stMotionStage.stAxisStatus.nCmdData:=INT_TO_UINT( stMotionStage.nCmdData);  //Or nCmdDataLocal
 stMotionStage.stAxisStatus.nCommand:=INT_TO_UINT( stMotionStage.nCommand);  //Or nCommandLocal
 stMotionStage.stAxisStatus.nErrorId:= stMotionStage.nErrorId;
 stMotionStage.stAxisStatus.bBusy:= stMotionStage.bBusy;
 stMotionStage.stAxisStatus.bHomed:= stMotionStage.bHomed;
 stMotionStage.stAxisStatus.bExecute:=bLocalExec;
 stMotionStage.stAxisStatus.nCommand:=3; // If this is not 3, the IOC stops updating positions during homing
END_METHOD

METHOD WriteParameterNC
VAR_INPUT
    Execute:BOOL;
    ParameterNumber : MC_AxisParameter;
    ParameterValue  : LREAL;
END_VAR
(*Do not change a moving axis parameter*)
fbMcWriteParameter(
    Axis:=stMotionStage.Axis,
    Execute:=(Execute AND stMotionStage.Axis.Status.NotMoving),
    ParameterNumber:=ParameterNumber,
    Value:=ParameterValue
);
END_METHOD

END_FUNCTION_BLOCK

(* stored: Version 1.1.0.1
   POU FB_MotionStageMCS2: Id {8a1beccb-8ae6-4cef-98b6-1d3261aefb9e}, SpecialFunc None
   Method ExposedParameters: Id {bfdcb735-2f35-43ca-9b4a-eca418143c19}
   Method FB_Init: Id {a8134580-303c-4b2f-8942-be52670189d3}
   Method Halt: Id {6287ad75-ad53-4d78-9e75-75537e8950c5}
   Method Interlock: Id {b0516fc0-3ac5-4a37-a4b7-b21194f9b805}
   Method MoveAbsolute: Id {c9986ba7-a025-4f1a-8312-93dc4112a24c}
   Method PersistParameters: Id {827e19b0-eb90-45f1-a0f0-e397f2f834ae}
   Method PostInit: Id {7af64fe1-72e2-4a67-9fd4-3933db27c0b4}
   Method PostMoveChecks: Id {20c015e9-bf00-4308-96ac-d493b364e91d}
   Method Power: Id {f641a677-a472-4a34-a0e0-f26f3662273e}
   Method Reset: Id {643b4736-0a43-4a18-8f6b-8a2439ed5e6f}
   Method RestoreMotionParams: Id {8335d215-fac8-43bf-97f2-e08acc164700}
   Method ScaleEncRawValue: Id {769f98a6-388a-461f-854a-93b1758d578f}
   Method SetEnables: Id {28f7e94e-bad4-40ca-b34a-f8da453343cc}
   Method UpdateEpicsStatus: Id {dc90c8f8-9d88-4ab9-9dc0-f90cd21b81fc}
   Method WriteParameterNC: Id {a04e1bd8-55ae-495c-bca4-be27f11603b4} *)
